Universal Robots URScript: 00C_06_JieXIan_ToZero.script

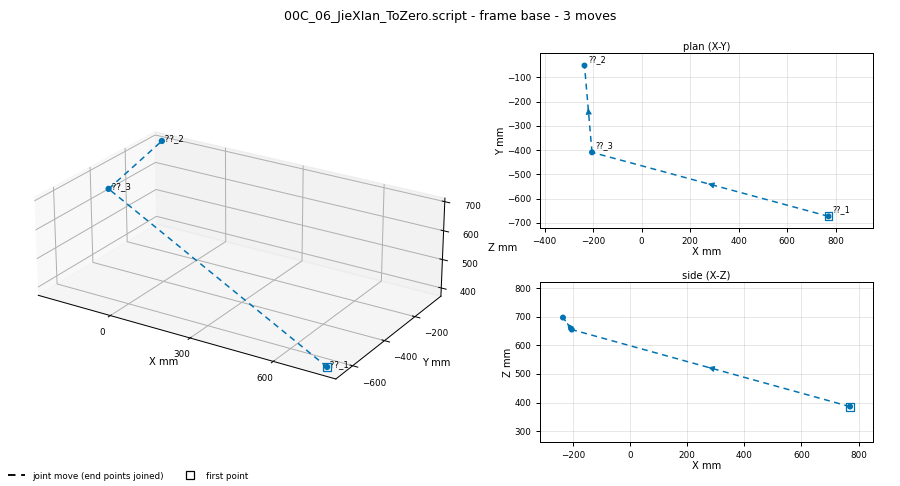
[picture p0: tool path of 00C_06_JieXIan_ToZero.script in frame base, 3 of 3 moves have a stored position in this frame; points joined in program order, loops and branches not executed]
def P00C_06_JieXIan_ToZero():
  set_gravity([0.0, 0.0, 9.82])
  set_safety_mode_transition_hardness(1)
  set_standard_analog_input_domain(0, 1)
  set_standard_analog_input_domain(1, 1)
  set_tool_analog_input_domain(0, 1)
  set_tool_analog_input_domain(1, 1)
  set_analog_outputdomain(0, 0)
  set_analog_outputdomain(1, 0)
  set_tool_voltage(24)
  set_input_actions_to_default()
  set_tcp(p[0.0,0.0,0.32,0.0,0.0,-0.5236])
  set_payload(8.0)
  global Zhua_1=[0.08063, -2.42649, -1.72682, -0.47876, 0.40808, -1.10831]
  global prepose=p[0.98979, -0.16931, -0.39963, 1.98720, 0.07234, 0.05469]
  global i_var_2=0
  global i_var_1=True
  global pose=p[0.98979, -0.31931, -0.39963, 1.98720, 0.07234, 0.05469]
  $ 1 "机器人程序"
  $ 2 "MoveJ"
  $ 3 "路点_1"
  set_tcp(p[-0.06262,0.03599,0.32923,0.0,0.0,1.3731])
  movej(get_inverse_kin(p[.770238853820, -.672649266252, .385667645850, .061502875430, -.012141238104, 1.533387331462], qnear=[-0.5369251410113733, -2.6996119658099573, -1.26943284669985, -0.7956278959857386, -1.5583685080157679, -0.8680942694293421]), a=0.6981317007977318, v=0.5235987755982988)
  $ 4 "路点_3"
  set_tcp(p[-0.06262,0.03599,0.32923,0.0,0.0,1.3731])
  movej(get_inverse_kin(p[-.204283704848, -.408876094608, .655327355532, .057445370057, -.016158455451, 1.700154836812], qnear=[-1.5327356497394007, -1.5895445982562464, -2.628538195286886, -0.5410311857806605, -1.602598015462057, 0.2885614037513733]), a=0.6981317007977318, v=0.5235987755982988)
  $ 5 "路点_2"
  set_tcp(p[-0.06262,0.03599,0.32923,0.0,0.0,1.3731])
  movej(get_inverse_kin(p[-.235273666055, -.051175590230, .697572943985, .005911176346, -.018034347169, 1.750475207962], qnear=[-1.5701916853534144, -2.1154085268193512E-4, -2.875479523335592, -1.853560749684469, -1.5660117308246058, 0.3727708160877228]), a=0.6981317007977318, v=0.5235987755982988)
end
